INTERFACE I_ReadableDisplayBuffer

METHOD PUBLIC TryReadPixel : BOOL;
VAR_INPUT
	X : DINT;
	Y : DINT;
	Pixel : REFERENCE TO Pixel;
END_VAR
END_METHOD

END_INTERFACE

(* stored: Version 1.1.0.1, ProductVersion 3.1.4024.15
   Itf I_ReadableDisplayBuffer: Id {2deb318d-7c62-4094-b7f2-b74403200da8}
   Method TryReadPixel: Id {b4078d39-9531-44f7-abe1-4048b65cb814} *)
